// SIMATIC S7-200 project (STEP 7-Micro/WIN), CPU 221 REL 01.10

SYMBOL_TABLE USR1
Always_On        SM0.0    // This bit is always on.
First_Scan_On    SM0.1    // This bit is on for the first scan cycle only.
PLS0_Ctrl        SMB67    // Controls pulse train output & pulse width modulation functions for output Q0.0.
PLS0_Cycle       SMW68    // Cycle time value, pulse train or pls. width modulation output 0. SMB68 is MSB.
PWM0_PW          SMW70    // Pulse width value of pulse width modulation output 0. SMB70 is the MSB.
Input_I0_0       I0.0     // Status of this input triggers interrupt events 0 (rising edge) or 1 (falling).
END_SYMBOL_TABLE

ORGANIZATION_BLOCK MAIN:OB1
TITLE=
// 题目：处理脉宽调制
// ***概述***
// 在S7-200系列中，CPU-214的输出端Q0.0和Q0.1能够输出方波信
// 号，而且方波信号的周期和脉宽均能独立调节，其中脉宽指的
// 是在一个周期内，输出信号处于高电平的时间长度
// 下面这个例子说明了脉宽调制（PWM）是如何工作的。输出端Q0.0输出方波信号，
// 其脉宽每周期递增0.5秒，周期固定为5秒，并且脉宽的初始值为0.5秒，当脉宽
// 达到设定的最大值4.5秒时，脉宽改为每周期递减0.5秒，直到脉宽为0为止，以
// 上过程周而复始
// 在这个例子中必须把输出端Q0.0与输入端I0.0连接，这样程序才能控制PWM。
// ***程序和注释***
// 特殊存储字节SMB67用来初始化输出端Q0.0的PWM.这个控制字内含PWM允许位，修
// 改周期和脉宽的允许位，以及时间基数选择位等，由子程序0来调整这个控制字节。
// 通过ENI指令，使所有的中断成为全局允许，然后通过PLS0指令，使系统接收各设定
// 值，并初始化“PTO/PWM发生器”从而在输出端Q0.0输出脉宽调制（PWM）信号。
// 另外，周期5秒是通过将数值5000置入特殊存储字SMW68来实现的，初始脉宽0.5
// 秒则通过将500写入特殊存储字SMW70来实现的。
// 这个初始化过程是在程序的第一个扫描周期通过子程序0来实现，第一个扫描周期
// 标志是SM0.1=1。当一个PWM循环结束，即当前脉宽为0秒时，将再一次初始化PWM。
// 辅助内存标记M0.0用来表明脉宽是增加还是减少，初始化时将这个标记设为增加。
// 输出端Q0.0与输入端I0.0相连,这样输出信号也可以送到输入端I0.0.当第一个方波
// 脉冲输出时，利用ATCH指令，把中断程序1（INT1）赋给中断事件0（I0.0的上升沿）
// 每个周期中断程序1将当前脉宽增加0.5秒，然后利用DTCH指令分离中断INT1,使这
// 个中断再次被屏蔽，如果在下次增加时，脉宽大于或等于周期，则将辅助内存标记
// 位M0.0再次置0。这样就把中断程序2赋予事件0，并且脉宽也将每次递减0.5秒。
//  当脉宽值减为0时，将再次执行，初始化程序（子程序0）
// 
BEGIN
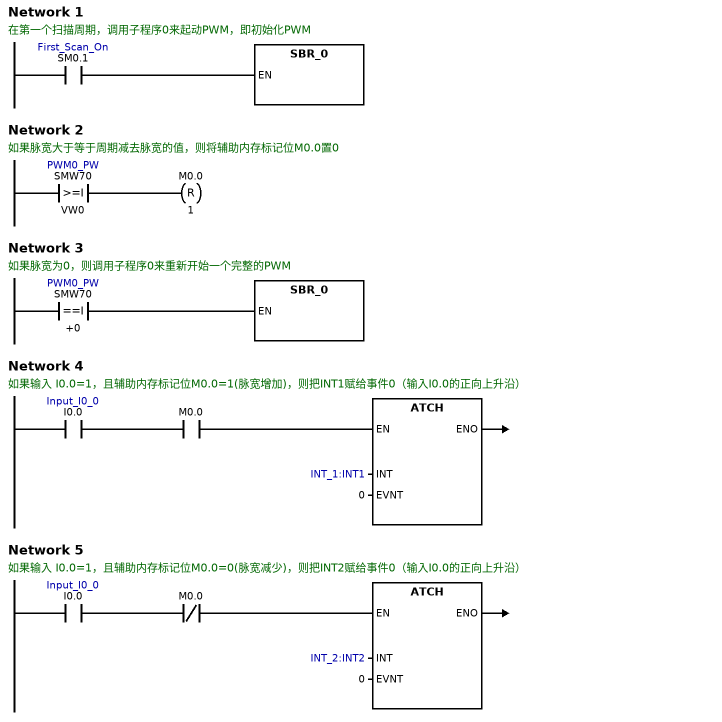
Network 1
// 在第一个扫描周期，调用子程序0来起动PWM，即初始化PWM
// 在第一个扫描周期SM0.1=1。
// 调用子程序0来起动PWM,即初始化PWM。
LD     First_Scan_On:SM0.1
CALL   SBR_0:SBR0
Network 2
// 如果脉宽大于等于周期减去脉宽的值，则将辅助内存标记位M0.0置0
//如果脉宽大于等于（周期-脉宽），
// 则将辅助内存标记位M0.0置0。
LDW>=  PWM0_PW:SMW70, VW0
R      M0.0, 1
Network 3
// 如果脉宽为0，则调用子程序0来重新开始一个完整的PWM
// 如果脉宽为0
// 则调用子程序0来重新开始一个完整的PWM
LDW=   PWM0_PW:SMW70, +0
CALL   SBR_0:SBR0
Network 4
// 如果输入 I0.0=1，且辅助内存标记位M0.0=1(脉宽增加)，则把INT1赋给事件0（输入I0.0的正向上升沿）
// 如果输入 I0.0=1
//且辅助内存标记位M0.0=1(脉宽增加)
//则把INT1赋给事件0（输入I0.0的正向上升沿）
LD     Input_I0_0:I0.0
A      M0.0
ATCH   INT_1:INT1, 0
Network 5
// 如果输入 I0.0=1，且辅助内存标记位M0.0=0(脉宽减少)，则把INT2赋给事件0（输入I0.0的正向上升沿）
// 如果输入 I0.0=1
// 且辅助内存标记位M0.0=0(脉宽减少)
//则把INT2赋给事件0（输入I0.0的正向上升沿）
LD     Input_I0_0:I0.0
AN     M0.0
ATCH   INT_2:INT2, 0
Network 6 //  主程序结束
// MEND				
// 
Network 7 // ***子程序0***
END_ORGANIZATION_BLOCK

SUBROUTINE_BLOCK SBR_0:SBR0
TITLE=
BEGIN
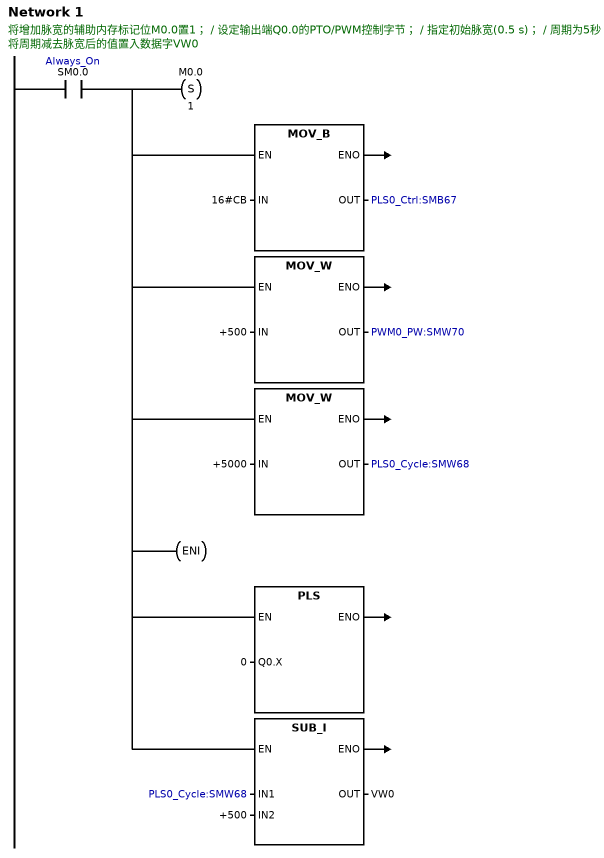
Network 1
// 将增加脉宽的辅助内存标记位M0.0置1；
// 设定输出端Q0.0的PTO/PWM控制字节；
// 指定初始脉宽(0.5 s)；
// 周期为5秒；
// 允许全部中断；
// 对PTO/PWM生成器编程的指令；
// 将周期置入数据字 VW0；
// 将周期减去脉宽后的值置入数据字VW0
// 将增加脉宽的辅助内存标记位M0.0置1
// 设定输出端Q0.0的PTO/PWM控制字节
// 指定初始脉宽(0.5 s).
// 周期为5秒
//允许全部中断
// 对PTO/PWM生成器编程的指令
//将周期置入数据字 VW0.
// 将（周期-脉宽）的值置入数据字VW0
LD     Always_On:SM0.0
S      M0.0, 1
MOVB   16#CB, PLS0_Ctrl:SMB67
MOVW   +500, PWM0_PW:SMW70
MOVW   +5000, PLS0_Cycle:SMW68
ENI
PLS    0
MOVW   PLS0_Cycle:SMW68, VW0
-I     +500, VW0
Network 2 //  子程序0结束并返回主程序
// RET				
// 
END_SUBROUTINE_BLOCK

INTERRUPT_BLOCK INT_1:INT1
TITLE=
BEGIN
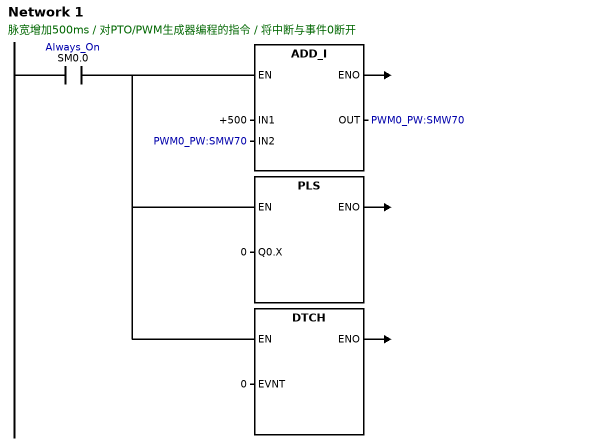
Network 1
// 脉宽增加500ms
// 对PTO/PWM生成器编程的指令
// 将中断与事件0断开
// 脉宽增加500ms
// 对PTO/PWM生成器编程的指令
//将中断与事件0断开
LD     Always_On:SM0.0
+I     +500, PWM0_PW:SMW70
PLS    0
DTCH   0
Network 2 //  中断服务程序1结束，并返回主程序
// RETI				
// 
END_INTERRUPT_BLOCK

INTERRUPT_BLOCK INT_2:INT2
TITLE=
BEGIN
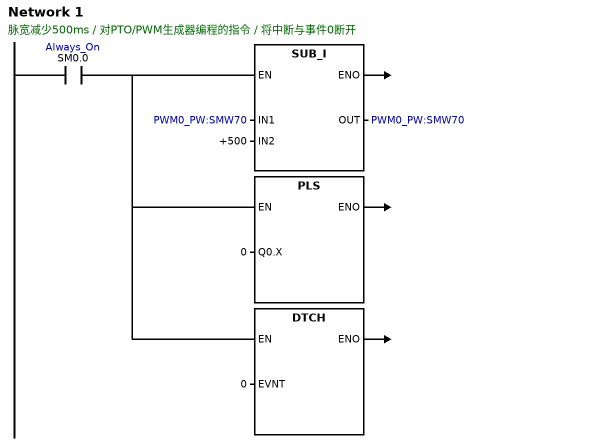
Network 1
// 脉宽减少500ms
// 对PTO/PWM生成器编程的指令
// 将中断与事件0断开
//  脉宽减少500ms
// 对PTO/PWM生成器编程的指令
//将中断与事件0断开
LD     Always_On:SM0.0
-I     +500, PWM0_PW:SMW70
PLS    0
DTCH   0
Network 2 // 中断服务程序2结束，并返回主程序
// RETI					
// 
END_INTERRUPT_BLOCK
